// TIA Portal V17 export
// export: Created 2023-12-22T15:28:30.5084901Z, ExportSetting WithDefaults, DisplayName Totally Integrated Automation Portal, DisplayVersion V17, DisplayName TIA Portal Openness, DisplayVersion V17, DisplayName TIA Portal Version Control Interface, DisplayVersion V17, DisplayName STEP 7 Professional, DisplayVersion V17, DisplayName STEP 7 Safety, DisplayVersion V17, DisplayName WinCC Advanced, DisplayVersion V17
FUNCTION_BLOCK "Historian"   // FB88, LAD
{ S7_Optimized_Access := 'FALSE' }
VERSION : 0.1
// stored: AutoNumber false, IsIECCheckEnabled false, SetENOAutomatically false, UDAEnableTagReadback false
   VAR_IN_OUT
      Main_REQ_Start : Bool;
      Main_Start : Bool;
      HMI_Start : Bool;
      HMI_Stop : Bool;
   END_VAR
   VAR DB_SPECIFIC
      pos : Array[0..15] of Bool;
      update : Bool;
      CMD : Bool;
      CODE : Int;
      DTL : DTL;
   END_VAR
   VAR
      LOG { S7_SetPoint := 'True'} : "Historian_LOG";
   END_VAR
   VAR CONSTANT
      tmp_x1 : Bool;
      tmp_x2 : Bool;
      tmp_x3 : Bool;
      any_conditions : Bool := true;
   END_VAR
   VAR_TEMP   // added for the SCL form of the ladder/FBD networks
      _w1 : Bool;
      _w2 : Bool;
      _w3 : Bool;
      _w4 : Bool;
   END_VAR
BEGIN

REGION Network 1: Запуск и останов с HMI
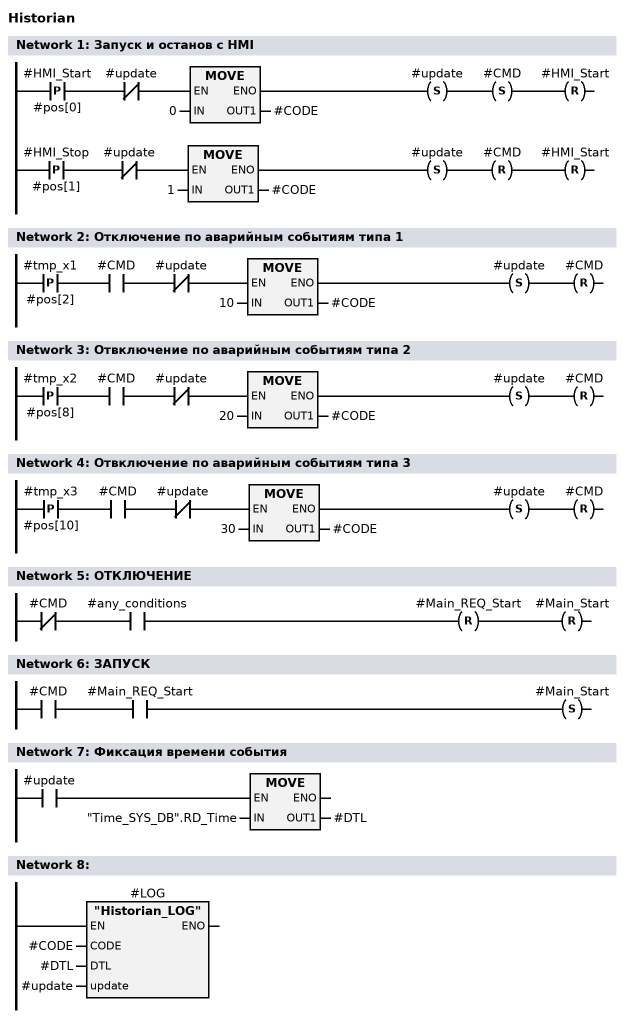
   RUNG wire#powerrail
      P_Contact(operand := #HMI_Start, bit := #pos[0])
      I_Contact( #update )
      Move(in := 0, out1 => #CODE)
      S_Coil( #update )
      S_Coil( #CMD )
      R_Coil( #HMI_Start )
   END_RUNG
   RUNG wire#powerrail
      P_Contact(operand := #HMI_Stop, bit := #pos[1])
      I_Contact( #update )
      Move(in := 1, out1 => #CODE)
      S_Coil( #update )
      R_Coil( #CMD )
      R_Coil( #HMI_Start )
   END_RUNG
   // the same network as SCL:
   #_w1 := #HMI_Start AND NOT #pos[0];   // rising edge of #HMI_Start
   #pos[0] := #HMI_Start;
   IF #_w1 AND NOT #update THEN #CODE := 0; END_IF;
   #_w2 := #_w1 AND NOT #update;
   IF #_w2 THEN
       #update := TRUE;
       #CMD := TRUE;
       #HMI_Start := FALSE;
   END_IF;
   #_w3 := #HMI_Stop AND NOT #pos[1];   // rising edge of #HMI_Stop
   #pos[1] := #HMI_Stop;
   IF #_w3 AND NOT #update THEN #CODE := 1; END_IF;
   #_w4 := #_w3 AND NOT #update;
   IF #_w4 THEN
       #update := TRUE;
       #CMD := FALSE;
       #HMI_Start := FALSE;
   END_IF;
END_REGION

REGION Network 2: Отключение по аварийным событиям типа 1
   RUNG wire#powerrail
      P_Contact(operand := #tmp_x1, bit := #pos[2])
      Contact( #CMD )
      I_Contact( #update )
      Move(in := 10, out1 => #CODE)
      S_Coil( #update )
      R_Coil( #CMD )
   END_RUNG
   // the same network as SCL:
   #_w1 := #tmp_x1 AND NOT #pos[2];   // rising edge of #tmp_x1
   #pos[2] := #tmp_x1;
   IF #_w1 AND #CMD AND NOT #update THEN #CODE := 10; END_IF;
   #_w2 := #_w1 AND #CMD AND NOT #update;
   IF #_w2 THEN
       #update := TRUE;
       #CMD := FALSE;
   END_IF;
END_REGION

REGION Network 3: Отвключение по аварийным событиям типа 2
   RUNG wire#powerrail
      P_Contact(operand := #tmp_x2, bit := #pos[8])
      Contact( #CMD )
      I_Contact( #update )
      Move(in := 20, out1 => #CODE)
      S_Coil( #update )
      R_Coil( #CMD )
   END_RUNG
   // the same network as SCL:
   #_w1 := #tmp_x2 AND NOT #pos[8];   // rising edge of #tmp_x2
   #pos[8] := #tmp_x2;
   IF #_w1 AND #CMD AND NOT #update THEN #CODE := 20; END_IF;
   #_w2 := #_w1 AND #CMD AND NOT #update;
   IF #_w2 THEN
       #update := TRUE;
       #CMD := FALSE;
   END_IF;
END_REGION

REGION Network 4: Отвключение по аварийным событиям типа 3
   RUNG wire#powerrail
      P_Contact(operand := #tmp_x3, bit := #pos[10])
      Contact( #CMD )
      I_Contact( #update )
      Move(in := 30, out1 => #CODE)
      S_Coil( #update )
      R_Coil( #CMD )
   END_RUNG
   // the same network as SCL:
   #_w1 := #tmp_x3 AND NOT #pos[10];   // rising edge of #tmp_x3
   #pos[10] := #tmp_x3;
   IF #_w1 AND #CMD AND NOT #update THEN #CODE := 30; END_IF;
   #_w2 := #_w1 AND #CMD AND NOT #update;
   IF #_w2 THEN
       #update := TRUE;
       #CMD := FALSE;
   END_IF;
END_REGION

REGION Network 5: ОТКЛЮЧЕНИЕ
   RUNG wire#powerrail
      I_Contact( #CMD )
      Contact( #any_conditions )
      R_Coil( #Main_REQ_Start )
      R_Coil( #Main_Start )
   END_RUNG
   // the same network as SCL:
   IF NOT #CMD AND #any_conditions THEN
       #Main_REQ_Start := FALSE;
       #Main_Start := FALSE;
   END_IF;
END_REGION

REGION Network 6: ЗАПУСК
   RUNG wire#powerrail
      Contact( #CMD )
      Contact( #Main_REQ_Start )
      S_Coil( #Main_Start )
   END_RUNG
   // the same network as SCL:
   IF #CMD AND #Main_REQ_Start THEN #Main_Start := TRUE; END_IF;
END_REGION

REGION Network 7: Фиксация времени события
   RUNG wire#powerrail
      Contact( #update )
      Move(in := "Time_SYS_DB".RD_Time, out1 => #DTL)
   END_RUNG
   // the same network as SCL:
   IF #update THEN #DTL := "Time_SYS_DB".RD_Time; END_IF;
END_REGION

REGION Network 8
   RUNG wire#powerrail
      #LOG(CODE := #CODE, DTL := #DTL, update := #update)
   END_RUNG
   // the same network as SCL:
   #LOG(CODE := #CODE, DTL := #DTL, update := #update);   // "Historian_LOG"
END_REGION
END_FUNCTION_BLOCK
